// SIMATIC STEP 7 (V5.x) project My_project_Adrian
// CPU: CPU 315-2 DP
// station: P_ADR_BUS
// station: Hardware
// station: Test_station
// station: P_ADR_BUS
// station: Configuration
// program: S7 Program(1)
// program: Day1

SYMBOL_TABLE
"Counter_Bay_1"	C 1	COUNTER	// Part counter for Bay 1
"Counter_Bay_2"	C 2	COUNTER	// Part counter for Bay 2
"Counter_Bay_3"	C 3	COUNTER	// Part counter for Bay 3
"Inst_DB_Bay_1_Counter"	DB 1	SFB 0
"Inst_DB_Bay_2_Counter"	DB 2	SFB 0
"Inst_DB_Bay_3_Counter"	DB 3	SFB 0
"Inst_DB_Belt_Fault"	DB 4	SFB 4
"DB_Data_Backup"	DB 10	DB 10	// Saves the production data every minute
"Instance_FB11"	DB 11	FB 11	// Instance DB for FB11
"Instance_FB12"	DB 12	FB 12	// Instance DB for FB12
"Instance_FB16"	DB 16	FB 16	// Instance DB for FB16
"Instance_FB18"	DB 18	FB 18	// Instance DB for FB 18
"DB_Weight_Values"	DB 30	DB 30
"Instance_FB42"	DB 42	FB 42	// Instance DB for FB42
"Instance_FB44"	DB 44	FB 44	// Instance DB for FB44
"DB_Data"	DB 50	DB 50	// Stores Data for FB42: MM420 Communication
"DB_LED_Status"	DB 51	DB 51	// Stores CPU LED Status
"DB_Diagnostic_data"	DB 86	DB 86	// Stores Profibus DP Slave errors
"DB_Area_Pointer"	DB 88	DB 88	// Stores HMI Area pointers
"DB_edge_detection"	DB 100	DB 100	// Stores edge detection flags
"FB_Running_light"	FB 11	FB 11	// Running light over 1 byte
"FB_Save_weight"	FB 12	FB 12
"FB_Conveyor"	FB 16	FB 16
"FB_Statistic"	FB 18	FB 18
"FB_MM420_PKW"	FB 42	FB 42	// shows PKW mechanism
"FB_MM420"	FB 44	FB 44	// Communciation with Micromaster
"FC_DT_TOD"	FC 8	FC 8	// DT to TOD
"FC_Supply_area_pointer"	FC 12	FC 12	// supply of the HMI area pointer
"FC_Signalization"	FC 14	FC 14	// Signalization
"FC_Modes"	FC 15	FC 15	// Mode selection
"FC_Conveyor"	FC 16	FC 16	// Control logic for conveyor belt
"FC_Statistic"	FC 18	FC 18	// Count parts
"FC_Production_Display"	FC 19	FC 19	// Display production data
"FC_Diagnostic"	FC 51	FC 51	// evaluation of SZL-sublists
"FC_Scale_Analog_value"	FC 105	FC 105	// Scaling block for analog value
"Heater_Timer"	FC 119	FC 119	// Activation of heater depending upon time of day
"T00 Start"	I 0.0	BOOL	// Pushbutton - System ON
"T01 Stop"	I 0.1	BOOL	// Pushbutton - System OFF
"T02 Jog right"	I 0.2	BOOL	// Pushbutton - Jog conveyor motor right
"T03 Jog left"	I 0.3	BOOL	// Pushbutton - Jog conveyor motor left
"T04 Auto/Man"	I 0.4	BOOL	// Mode selector switch Man/Auto 0""/""1""""
"T05 Accept_Mode"	I 0.5	BOOL	// Pushbutton - Accept mode selection
"T06 Ack. Faults"	I 0.6	BOOL	// Fault Acknowledgement
"T07 Delete Memory"	I 0.7	BOOL	// Deletes the Statistic Memory
"T10 Ack_Fault"	I 1.0	BOOL	// Fault acknowledgement switch
"Analog_Store_Start"	I 1.5	BOOL	// Initiate storage of analog values into DB30
"T16_Ack_Analog_Alarm"	I 1.6	BOOL	// Reset analog HI/LO alarm
"T17_Acknowledge_Startup"	I 1.7	BOOL	// Pushbutton for startup acknowledgement
"LB1"	I 8.0	BOOL	// Light barrier at conveyor end
"T_PB1"	I 8.1	BOOL	// Acknowledge PB at Bay 1
"T_PB2"	I 8.2	BOOL	// Acknowledge PB at Bay 2
"T_PB3"	I 8.3	BOOL	// Acknowledge PB at Bay 3
"T_PB4"	I 8.4	BOOL	// Acknowledge PB at Bay 4
"BAY1"	I 8.5	BOOL	// Proximity Switch 01 for Bay1 (INI1)
"BAY2"	I 8.6	BOOL	// Proximity Switch 02 for Bay2 (INI2)
"BAY3"	I 8.7	BOOL	// Proximity Switch 03 for Bay3 (INI3)
"LB_ET"	I 88.0	BOOL
"T_PB1_ET"	I 88.1	BOOL
"T_PB2_ET"	I 88.2	BOOL
"T_PB3_ET"	I 88.3	BOOL
"T_PB4_ET"	I 88.4	BOOL
"BAY1_ET"	I 88.5	BOOL	// Proximity Switch 01 for Bay1 (INI1)
"BAY2_ET"	I 88.6	BOOL	// Proximity Switch 02 for Bay2 (INI2)
"BAY3_ET"	I 88.7	BOOL	// Proximity Switch 03 for Bay3 (INI3)
"IW_BCD"	IW 2	WORD	// BCD Thumbwheel, presets
"Always_Off"	M 0.0	BOOL	// Bit reset in OB100 at start-up
"Always_On"	M 0.1	BOOL	// Bit set in OB100 at start-up
"M_Flash_10Hz"	M 10.0	BOOL	// Memory bit - flashing frequency 10Hz
"M_Flash_2Hz"	M 10.3	BOOL	// Memory bit - flashing frequency 2Hz
"Delay_lockout"	M 14.0	BOOL	// Lockout conveyor movement after 6 seconds
"K_LT_Manual_Mode"	M 16.0	BOOL	// Conveyor runs in Manual mode
"K_LT_Auto_Mode"	M 16.1	BOOL	// Conveyor runs in Auto mode
"M_Motor_ON"	M 31.0	BOOL	// Request: Motor On
"M_Weight_OK"	M 35.0	BOOL	// Weight value is within tolerance
"M_Analog_module_error"	M 40.0	BOOL
"M_Motor_Stop"	M 46.0	BOOL	// Motor stop PB on HMI screen
"Weight_OK_Edge"	M 50.3	BOOL	// Edge storage bit for weight within tolerance message
"Weight_Not_OK_Edge"	M 50.4	BOOL	// Edge storage bit for weight outside tolerance message
"Weight_Scaled_REAL"	MD 70	REAL	// Current weight on the scale (REAL)
"Frequency_Required"	MD 130	REAL	// Enter required frequency setpoint
"Ramp_Up_Time"	MD 136	REAL	// Ramp up time value in seconds
"Ramp_Down_Time"	MD 140	REAL	// Ramp down time value in seconds
"Motor_Request"	MW 44	INT	// Command list number from HMI screen
"Quantity_Bay_1"	MW 100	INT	// Number of parts counted at Bay 1
"Quantity_Bay_2"	MW 102	INT	// Number of parts counted at Bay 2
"Quantity_Bay_3"	MW 104	INT	// Number of parts counted at Bay 3
"Total_Quantity"	MW 106	INT	// Sum of all parts counted
"Utilisation_Bay_1"	MW 110	INT	// % utilisation of bay 1
"Utilisation_Bay_2"	MW 112	INT	// % utilisation of bay 2
"Utilisation_Bay_3"	MW 114	INT	// % utilisation of bay 3
"Parameter_Number"	MW 134	INT	// Enter number of parameter to change
"CYCL_EXC"	OB 1	OB 1	// Cycle Execution
"OB_Time_Interrupt"	OB 10	OB 10
"OB_Check Weight"	OB 35	OB 35
"OB_Hardware_Interrupt"	OB 40	OB 40
"I/O_FLT1"	OB 82	OB 82	// I/O Point Fault 1
"OB_RACK_FLT"	OB 86	OB 86	// Loss of Rack Fault
"OB_Startup"	OB 100	OB 100	// automatic or manual restart
"PROG_ERR"	OB 121	OB 121	// Programming Error
"OB_Periph_Error"	OB 122	OB 122
"Status_Word_MM420"	PIW 256	WORD	// Status word from MM420 drive (feedback)
"Actual_Speed_MM420"	PIW 258	WORD	// Actual speed from MM420 drive (feedback)
"Analog_Channel_1"	PIW 304	INT	// Analog channel 1 (Potentiometer)
"Control_Word_MM420"	PQW 256	WORD	// Control word for the MM420 AC drive
"Setpoint_Speed_MM420"	PQW 258	WORD	// Setpoint speed for the MM420
"L_Belt_fault"	Q 4.0	BOOL	// Indicator light - conveyor belt fault condition
"L_SYSTEM"	Q 4.1	BOOL	// Indicator light - System ON
"L_Mode_MANUAL"	Q 4.2	BOOL	// Indicator light - MANUAL Mode ON
"L_Mode_AUTO"	Q 4.3	BOOL	// Indicator light - AUTO Mode ON
"L_Restart_M"	Q 4.5	BOOL	// Indicator light, manual restart
"L_Restart_A"	Q 4.6	BOOL	// Indicator light, auto restart
"L_Weight_not_okay"	Q 5.1	BOOL	// Indicator - weight not within tolerance
"L_Analog_Limit_Alarm"	Q 5.2	BOOL	// Analog channel has exceeded voltage limits
"Heater"	Q 5.3	BOOL	// Heater
"L_Bay1"	Q 8.1	BOOL	// Indicator light - Bay 1 (H1)
"L_Bay2"	Q 8.2	BOOL	// Indicator light - Bay 2 (H2)
"L_Bay3"	Q 8.3	BOOL	// Indicator light - Bay 3 (H3)
"L4_Preassembly"	Q 8.4	BOOL	// Indicator light - Preassembly (H4)
"K_RT"	Q 8.5	BOOL	// Contactor for Conveyor Belt move RIGHT
"K_LT"	Q 8.6	BOOL	// Contactor for Conveyor Belt move LEFT
"Horn"	Q 8.7	BOOL	// Signal on Conveyor
"L_Bay1_ET"	Q 88.1	BOOL	// Indicator light - Bay 1 (H1) into ET200S
"L_Bay2_ET"	Q 88.2	BOOL	// Indicator light - Bay 2 (H2) into ET200S
"L_Bay3_ET"	Q 88.3	BOOL	// Indicator light - Bay 3 (H3) into ET200S
"L4_Preassembly_ET"	Q 88.4	BOOL	// Indicator light - Preassembly (H4) into ET200S
"K_RT_ET"	Q 88.5	BOOL	// Contactor for Conveyor Belt move RIGHT into ET200S
"K_LT_ET"	Q 88.6	BOOL	// Contactor for Conveyor Belt move LEFT into ET200S
"Horn_ET"	Q 88.7	BOOL	// Signal on Conveyor into ET200S
"Running_Lights"	QB 8	BYTE	// Output LED's running indicate start-up has occured
"MM420_PZD"	QD 56	DWORD	// Control and main setpoint of MM420
"QW_Display"	QW 6	WORD	// Binary Coded Decimal (BCD) number display
"CTU"	SFB 0	SFB 0	// Count Up
"TON"	SFB 4	SFB 4	// Generate an On Delay
"TOF"	SFB 5	SFB 5	// Generate an Off Delay
"READ_CLK"	SFC 1	SFC 1	// Read System Clock
"DPRD_DAT"	SFC 14	SFC 14	// Read Consistent Data of a Standard DP Slave
"DPWR_DAT"	SFC 15	SFC 15	// Write Consistent Data to a Standard DP Slave
"BLKMOV"	SFC 20	SFC 20	// Copy Variables
"FILL"	SFC 21	SFC 21	// Initialize a Memory Area
"STP"	SFC 46	SFC 46	// Change the CPU to STOP
"RDSYSST"	SFC 51	SFC 51	// Read a System Status List or Partial List
"WR_USMSG"	SFC 52	SFC 52	// Write a User-Defined Diagnostic Event to the Diagnostic Buffer
"Right_Lockout_Timer"	T 1	TIMER	// 2 s lockout timer for right direction
"Left_Lockout_Timer"	T 2	TIMER	// 2 s lockout timer for left direction
"SD_Runtime_error"	T 14	TIMER	// Transport monitoring
"SD_Startup_delay"	T 16	TIMER	// Conveyor starts in Auto mode after a delay
"CPU_LED_Record"	UDT 51	UDT 51	// CPU LED information
"Conveyor_Model"	VAT 1	
"VAT_18"	VAT 2	
"VAT_FB42"	VAT 3	
END_SYMBOL_TABLE

FUNCTION_BLOCK "FB_Running_light"	// FB 11
VERSION : 0.1
VAR_INPUT
  Flash_frequency : BOOL ;
  Restart : BOOL ;
END_VAR
VAR_OUTPUT
  Running_light : BYTE ;
END_VAR
VAR
  EM_flash : BOOL ;
  EM_restart : BOOL ;
END_VAR
BEGIN
NETWORK
TITLE =
      A     #Restart;
      FP    #EM_restart;
      JCN   next;
      L     1;
      T     #Running_light;
NETWORK
TITLE =
next: A     #Restart;
      JCN   end;
      A     #Flash_frequency;
      FP    #EM_flash;
      JCN   end;
      L     #Running_light;
      SLW   1;
      L     128;
      >I;
      TAK;
      JCN   rett;
      L     1;
rett: T     #Running_light;
end:  NOP   0;
END_FUNCTION_BLOCK

FUNCTION "FC_Signalization" : VOID	// FC 14
VERSION : 0.1
BEGIN
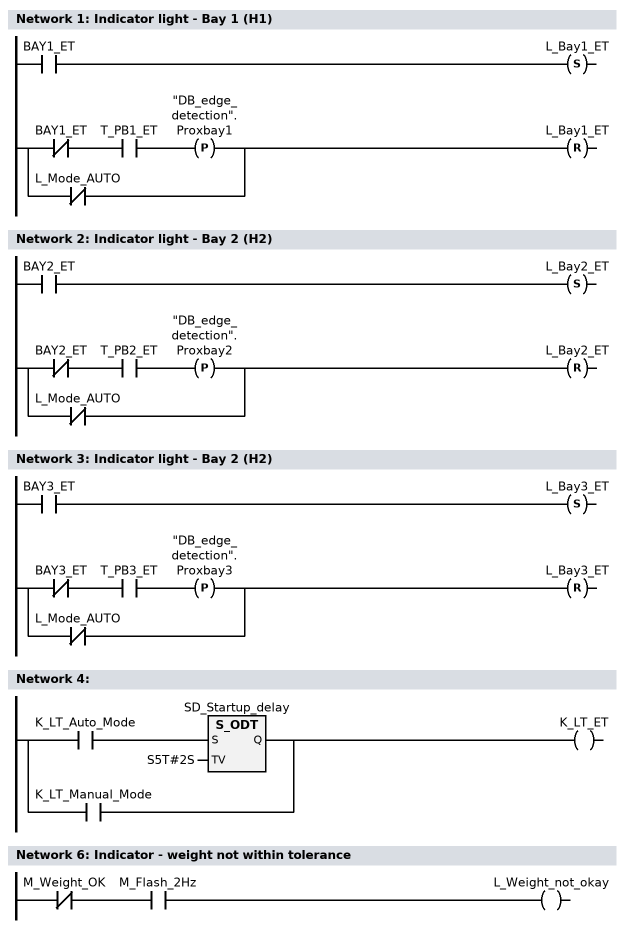
NETWORK
TITLE = Indicator light - Bay 1 (H1)
      A     "BAY1_ET";
      S     "L_Bay1_ET";
      A(;
      AN    "BAY1_ET";
      A(;
      A     "T_PB1_ET";
      BLD   100;
      FP    "DB_edge_detection".Proxbay1;
      );
      ON    "L_Mode_AUTO";
      );
      R     "L_Bay1_ET";
      NOP   0;
NETWORK
TITLE = Indicator light - Bay 2 (H2)
      A     "BAY2_ET";
      S     "L_Bay2_ET";
      A(;
      AN    "BAY2_ET";
      A(;
      A     "T_PB2_ET";
      BLD   100;
      FP    "DB_edge_detection".Proxbay2;
      );
      ON    "L_Mode_AUTO";
      );
      R     "L_Bay2_ET";
      NOP   0;
NETWORK
TITLE = Indicator light - Bay 2 (H2)
      A     "BAY3_ET";
      S     "L_Bay3_ET";
      A(;
      AN    "BAY3_ET";
      A(;
      A     "T_PB3_ET";
      BLD   100;
      FP    "DB_edge_detection".Proxbay3;
      );
      ON    "L_Mode_AUTO";
      );
      R     "L_Bay3_ET";
      NOP   0;
NETWORK
TITLE =
      O(;
      A     "K_LT_Auto_Mode";
      L     S5T#2S;
      SD    "SD_Startup_delay";
      NOP   0;
      NOP   0;
      NOP   0;
      A     "SD_Startup_delay";
      );
      O     "K_LT_Manual_Mode";
      =     "K_LT_ET";
NETWORK
TITLE =
      A(;
      A(;
      A     "K_LT_ET";
      A     "L_Restart_A";
      L     S5T#6S;
      SD    "SD_Runtime_error";
      NOP   0;
      NOP   0;
      NOP   0;
      A     "SD_Runtime_error";
      );
      S     "Delay_lockout";
      A(;
      A     "T10 Ack_Fault";
      BLD   100;
      FP    "DB_edge_detection".UNNAMED;
      );
      R     "Delay_lockout";
      A     "Delay_lockout";
      );
      A     "M_Flash_2Hz";
      =     "L_Belt_fault";
NETWORK
TITLE = Indicator - weight not within tolerance
      AN    "M_Weight_OK";
      A     "M_Flash_2Hz";
      =     "L_Weight_not_okay";
END_FUNCTION

FUNCTION "FC_Modes" : VOID	// FC 15
VERSION : 0.1
BEGIN
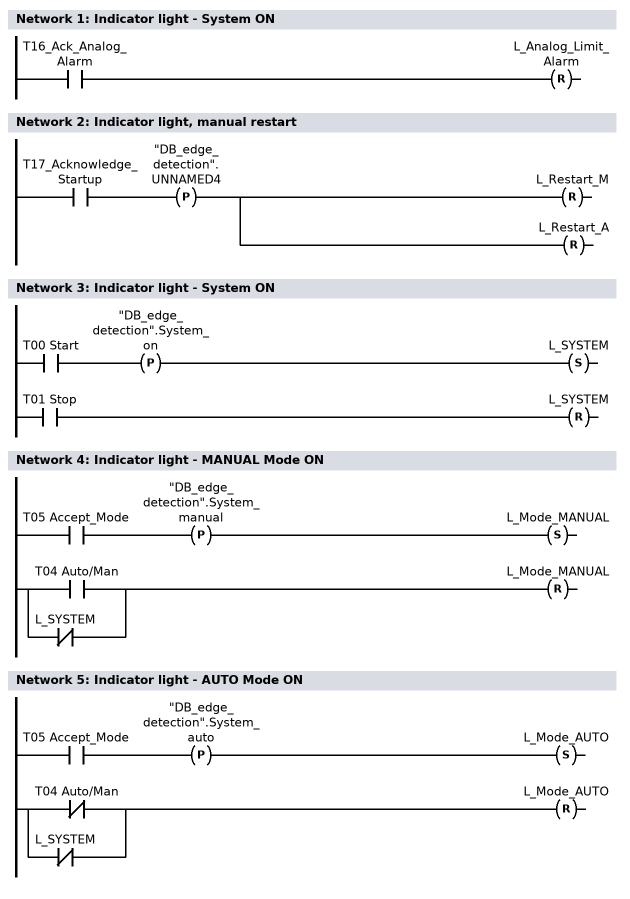
NETWORK
TITLE = Indicator light - System ON
      A     "T16_Ack_Analog_Alarm";
      R     "L_Analog_Limit_Alarm";
NETWORK
TITLE = Indicator light, manual restart
      A     "T17_Acknowledge_Startup";
      BLD   100;
      FP    "DB_edge_detection".UNNAMED4;
      R     "L_Restart_M";
      R     "L_Restart_A";
NETWORK
TITLE = Indicator light - System ON
      A     "T00 Start";
      FP    "DB_edge_detection".System_on;
      S     "L_SYSTEM";
      A     "T01 Stop";
      R     "L_SYSTEM";
      NOP   0;
NETWORK
TITLE = Indicator light - MANUAL Mode ON
      A     "T05 Accept_Mode";
      FP    "DB_edge_detection".System_manual;
      S     "L_Mode_MANUAL";
      A(;
      O     "T04 Auto/Man";
      ON    "L_SYSTEM";
      );
      R     "L_Mode_MANUAL";
      NOP   0;
NETWORK
TITLE = Indicator light - AUTO Mode ON
      A     "T05 Accept_Mode";
      FP    "DB_edge_detection".System_auto;
      S     "L_Mode_AUTO";
      A(;
      ON    "T04 Auto/Man";
      ON    "L_SYSTEM";
      );
      R     "L_Mode_AUTO";
      NOP   0;
END_FUNCTION

FUNCTION "FC_Conveyor" : VOID	// FC 16
VERSION : 0.1
BEGIN
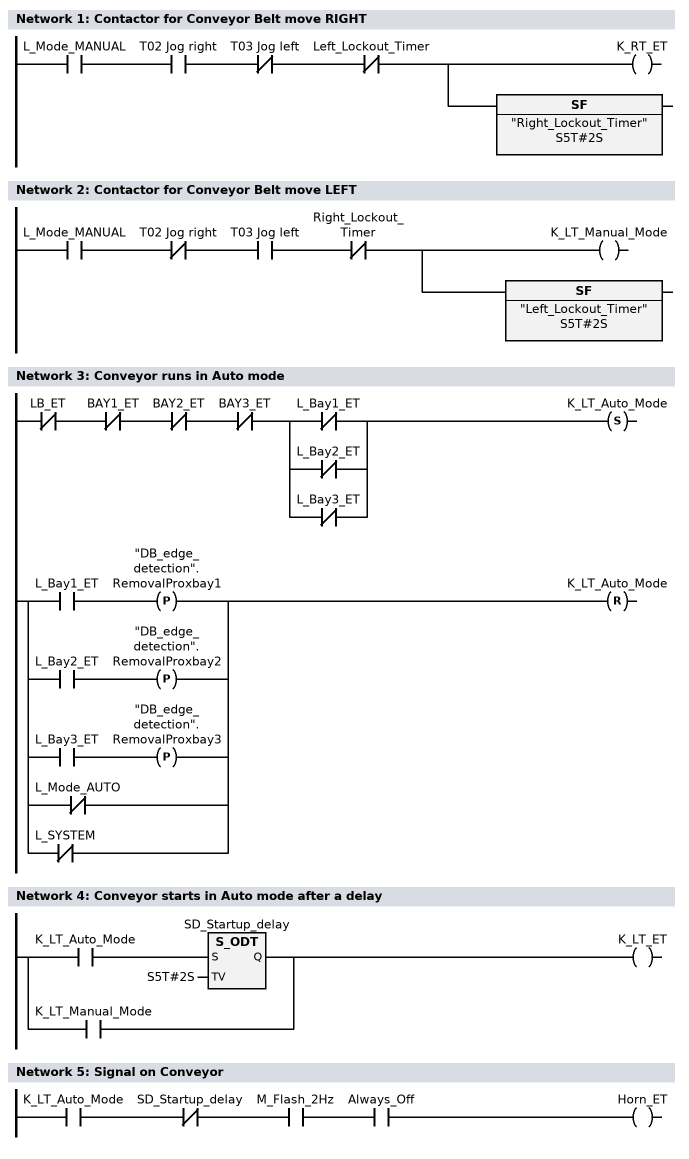
NETWORK
TITLE = Contactor for Conveyor Belt move RIGHT
      A     "L_Mode_MANUAL";
      A     "T02 Jog right";
      AN    "T03 Jog left";
      AN    "Left_Lockout_Timer";
      =     "K_RT_ET";
      L     S5T#2S;
      SF    "Right_Lockout_Timer";
NETWORK
TITLE = Contactor for Conveyor Belt move LEFT
      A     "L_Mode_MANUAL";
      AN    "T02 Jog right";
      A     "T03 Jog left";
      AN    "Right_Lockout_Timer";
      =     "K_LT_Manual_Mode";
      L     S5T#2S;
      SF    "Left_Lockout_Timer";
NETWORK
TITLE = Conveyor runs in Auto mode
      AN    "LB_ET";
      AN    "BAY1_ET";
      AN    "BAY2_ET";
      AN    "BAY3_ET";
      A(;
      ON    "L_Bay1_ET";
      ON    "L_Bay2_ET";
      ON    "L_Bay3_ET";
      );
      S     "K_LT_Auto_Mode";
      A(;
      A     "L_Bay1_ET";
      FP    "DB_edge_detection".RemovalProxbay1;
      O(;
      A     "L_Bay2_ET";
      FP    "DB_edge_detection".RemovalProxbay2;
      );
      O(;
      A     "L_Bay3_ET";
      FP    "DB_edge_detection".RemovalProxbay3;
      );
      ON    "L_Mode_AUTO";
      ON    "L_SYSTEM";
      );
      R     "K_LT_Auto_Mode";
      NOP   0;
NETWORK
TITLE = Conveyor starts in Auto mode after a delay
      O(;
      A     "K_LT_Auto_Mode";
      L     S5T#2S;
      SD    "SD_Startup_delay";
      NOP   0;
      NOP   0;
      NOP   0;
      A     "SD_Startup_delay";
      );
      O     "K_LT_Manual_Mode";
      =     "K_LT_ET";
NETWORK
TITLE = Signal on Conveyor
      A     "K_LT_Auto_Mode";
      AN    "SD_Startup_delay";
      A     "M_Flash_2Hz";
      A     "Always_Off";
      =     "Horn_ET";
END_FUNCTION

FUNCTION "FC_Statistic" : VOID	// FC 18
VERSION : 0.1
VAR_TEMP
  aux_Real : REAL ;
END_VAR
BEGIN
NETWORK
TITLE =
      A     "L_Bay1_ET";
      =     L 4.0;
      BLD   103;
      A     "T07 Delete Memory";
      FP    "DB_edge_detection".UNNAMED1;
      =     L 4.1;
      BLD   103;
      BLD   9;
      =     L 9.0;
      CDB;
      OPN   DI 1;
      TAR2  LD 5;
      A     L 4.0;
      =     DIX 0.0;
      A     L 4.1;
      =     DIX 0.1;
      LAR2  P#DBX 0.0;
      UC    "CTU";
      LAR2  LD 5;
      L     DIW 6;
      T     "Quantity_Bay_1";
      CDB;
      BLD   10;
      NOP   0;
NETWORK
TITLE = Part counter for Bay 2
      A     "L_Bay2_ET";
      =     L 4.0;
      BLD   103;
      A     "T07 Delete Memory";
      FP    "DB_edge_detection".UNNAMED2;
      =     L 4.1;
      BLD   103;
      BLD   9;
      =     L 9.0;
      CDB;
      OPN   DI 2;
      TAR2  LD 5;
      A     L 4.0;
      =     DIX 0.0;
      A     L 4.1;
      =     DIX 0.1;
      LAR2  P#DBX 0.0;
      UC    "CTU";
      LAR2  LD 5;
      L     DIW 6;
      T     "Quantity_Bay_2";
      CDB;
      BLD   10;
      NOP   0;
NETWORK
TITLE = Part counter for Bay 1
      A     "L_Bay3_ET";
      =     L 4.0;
      BLD   103;
      A     "T07 Delete Memory";
      FP    "DB_edge_detection".UNNAMED2;
      =     L 4.1;
      BLD   103;
      BLD   9;
      =     L 9.0;
      CDB;
      OPN   DI 3;
      TAR2  LD 5;
      A     L 4.0;
      =     DIX 0.0;
      A     L 4.1;
      =     DIX 0.1;
      LAR2  P#DBX 0.0;
      UC    "CTU";
      LAR2  LD 5;
      L     DIW 6;
      T     "Quantity_Bay_3";
      CDB;
      BLD   10;
      NOP   0;
NETWORK
TITLE =
      L     "Quantity_Bay_1";
      L     "Quantity_Bay_2";
      +I;
      L     "Quantity_Bay_3";
      +I;
      T     "Total_Quantity";
NETWORK
TITLE =
      L     "Total_Quantity";
      ITD;
      DTR;
      T     #aux_Real;
NETWORK
TITLE =
      L     "Total_Quantity";
      L     0;
      ==I;
      JCN   END1;
      L     0;
      T     "Utilisation_Bay_1";
      L     0;
      T     "Utilisation_Bay_1";
      T     "Utilisation_Bay_2";
      T     "Utilisation_Bay_3";
      BEU;
END1: NOP   0;
NETWORK
TITLE =
      L     "Quantity_Bay_1";
      ITD;
      DTR;
      L     1.000000e+02;
      *R;
      L     #aux_Real;
      /R;
      RND;
      T     "Utilisation_Bay_1";
NETWORK
TITLE =
      L     "Quantity_Bay_2";
      ITD;
      DTR;
      L     1.000000e+02;
      *R;
      L     #aux_Real;
      /R;
      RND;
      T     "Utilisation_Bay_2";
NETWORK
TITLE =
      L     "Quantity_Bay_3";
      ITD;
      DTR;
      L     1.000000e+02;
      *R;
      L     #aux_Real;
      /R;
      RND;
      T     "Utilisation_Bay_3";
END_FUNCTION

FUNCTION "FC_Production_Display" : VOID	// FC 19
VERSION : 0.1
VAR_INPUT
  Selection : WORD ;
END_VAR
VAR_OUTPUT
  Display : WORD ;
END_VAR
BEGIN
NETWORK
TITLE =
      L     #Selection;
      BTI;
      AW    W#16#F;
      DEC   1;
      JL    out;
      JU    bay1;
      JU    bay2;
      JU    bay3;
      JU    tot;
      JU    ut1;
      JU    ut2;
      JU    ut3;
      JU    wght;
out:  L     W#16#EEEE;
      JU    tran;
bay1: L     "Quantity_Bay_1";
      JU    anz;
bay2: L     "Quantity_Bay_2";
      JU    anz;
bay3: L     "Quantity_Bay_3";
      JU    anz;
tot:  L     "Total_Quantity";
      JU    anz;
ut1:  L     "Utilisation_Bay_1";
      JU    anz;
ut2:  L     "Utilisation_Bay_2";
      JU    anz;
ut3:  L     "Utilisation_Bay_3";
      JU    anz;
wght: L     "Weight_Scaled_REAL";
      TRUNC;
      DTB;
anz:  ITB;
tran: T     #Display;
END_FUNCTION

// FC 105: know-how protected block, not included

DATA_BLOCK "Inst_DB_Bay_1_Counter"	// DB 1
AUTHOR : SIMATIC
FAMILY : IEC_TC
VERSION : 0.0
"CTU"
BEGIN
END_DATA_BLOCK

DATA_BLOCK "Inst_DB_Bay_2_Counter"	// DB 2
AUTHOR : SIMATIC
FAMILY : IEC_TC
VERSION : 0.0
"CTU"
BEGIN
END_DATA_BLOCK

DATA_BLOCK "Inst_DB_Bay_3_Counter"	// DB 3
AUTHOR : SIMATIC
FAMILY : IEC_TC
VERSION : 0.0
"CTU"
BEGIN
END_DATA_BLOCK

DATA_BLOCK "DB_Data_Backup"	// DB 10
VERSION : 0.1
  STRUCT
   BAY : ARRAY  [1 .. 3 ] OF //counting partsfor every bay
   INT  := 0;
   Total_quantity : INT ;	//total summary
   Dummy : INT ;	//Dummy address
   Production_capacity : ARRAY  [1 .. 3 ] OF //Production capacity
   INT  := 0;
  END_STRUCT ;	
BEGIN
END_DATA_BLOCK

DATA_BLOCK "Instance_FB11"	// DB 11
VERSION : 0.0
"FB_Running_light"
BEGIN
END_DATA_BLOCK

DATA_BLOCK "DB_edge_detection"	// DB 100
VERSION : 0.1
  STRUCT
   System_on : BOOL ;
   System_manual : BOOL ;
   System_auto : BOOL ;
   Proxbay1 : BOOL ;
   Proxbay2 : BOOL ;
   Proxbay3 : BOOL ;
   RemovalProxbay1 : BOOL ;
   RemovalProxbay2 : BOOL ;
   RemovalProxbay3 : BOOL ;
   UNNAMED : BOOL ;	//Temporary placeholder variable
   UNNAMED1 : BOOL ;	//Temporary placeholder variable
   UNNAMED2 : BOOL ;	//Temporary placeholder variable
   UNNAMED3 : BOOL ;	//Temporary placeholder variable
   UNNAMED4 : BOOL ;	//Temporary placeholder variable
   UNNAMED5 : BOOL ;	//Temporary placeholder variable
   UNNAMED6 : BOOL ;	//Temporary placeholder variable
   UNNAMED7 : BOOL ;	//Temporary placeholder variable
   UNNAMED8 : BOOL ;	//Temporary placeholder variable
   UNNAMED9 : BOOL ;	//Temporary placeholder variable
   UNNAMED10 : BOOL ;	//Temporary placeholder variable
   UNNAMED11 : BOOL ;	//Temporary placeholder variable
   UNNAMED12 : BOOL ;	//Temporary placeholder variable
   UNNAMED13 : BOOL ;	//Temporary placeholder variable
   UNNAMED14 : BOOL ;	//Temporary placeholder variable
   UNNAMED15 : BOOL ;	//Temporary placeholder variable
   UNNAMED16 : BOOL ;	//Temporary placeholder variable
   UNNAMED17 : BOOL ;	//Temporary placeholder variable
   UNNAMED18 : BOOL ;	//Temporary placeholder variable
   UNNAMED19 : BOOL ;	//Temporary placeholder variable
   UNNAMED20 : BOOL ;	//Temporary placeholder variable
   UNNAMED21 : BOOL ;	//Temporary placeholder variable
   UNNAMED22 : BOOL ;	//Temporary placeholder variable
   UNNAMED23 : BOOL ;	//Temporary placeholder variable
   UNNAMED24 : BOOL ;	//Temporary placeholder variable
  END_STRUCT ;	
BEGIN
END_DATA_BLOCK

ORGANIZATION_BLOCK "CYCL_EXC"	// OB 1
TITLE = "Main Program Sweep (Cycle)"
VERSION : 0.1
VAR_TEMP
  OB1_EV_CLASS : BYTE ;	//Bits 0-3 = 1 (Coming event), Bits 4-7 = 1 (Event class 1)
  OB1_SCAN_1 : BYTE ;	//1 (Cold restart scan 1 of OB 1), 3 (Scan 2-n of OB 1)
  OB1_PRIORITY : BYTE ;	//Priority of OB Execution
  OB1_OB_NUMBR : BYTE ;	//1 (Organization block 1, OB1)
  OB1_RESERVED_1 : BYTE ;	//Reserved for system
  OB1_RESERVED_2 : BYTE ;	//Reserved for system
  OB1_PREV_CYCLE : INT ;	//Cycle time of previous OB1 scan (milliseconds)
  OB1_MIN_CYCLE : INT ;	//Minimum cycle time of OB1 (milliseconds)
  OB1_MAX_CYCLE : INT ;	//Maximum cycle time of OB1 (milliseconds)
  OB1_DATE_TIME : DATE_AND_TIME ;	//Date and time OB1 started
END_VAR
BEGIN
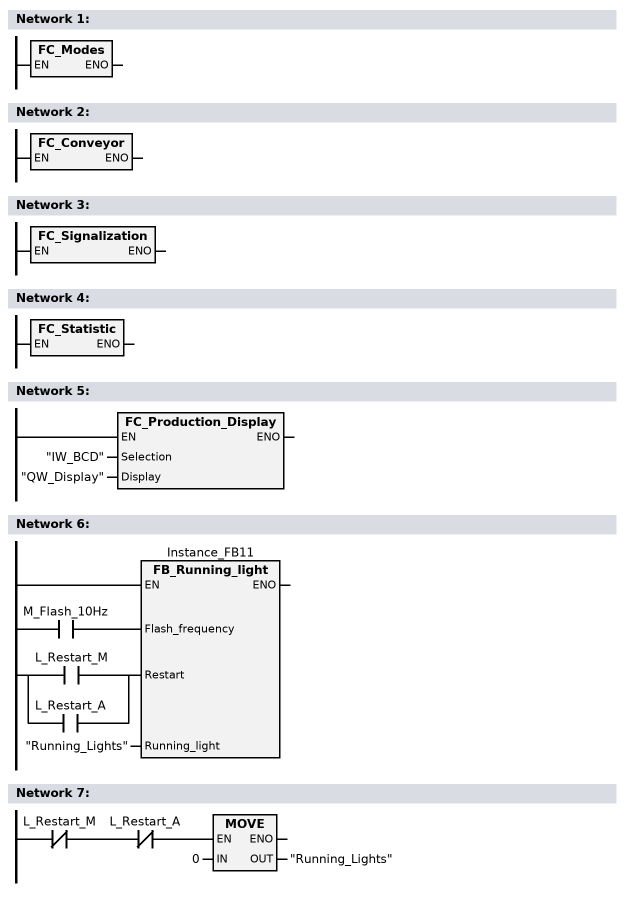
NETWORK
TITLE =
      CALL  "FC_Modes";
      NOP   0;
NETWORK
TITLE =
      CALL  "FC_Conveyor";
      NOP   0;
NETWORK
TITLE =
      CALL  "FC_Signalization";
      NOP   0;
NETWORK
TITLE =
      CALL  "FC_Statistic";
      NOP   0;
NETWORK
TITLE =
      CALL  "FC_Production_Display" (
           Selection                := "IW_BCD",
           Display                  := "QW_Display");
      NOP   0;
NETWORK
TITLE =
      A     "M_Flash_10Hz";
      =     L 20.0;
      BLD   103;
      A(;
      O     "L_Restart_M";
      O     "L_Restart_A";
      );
      =     L 20.1;
      BLD   103;
      CALL  "FB_Running_light" , "Instance_FB11" (
           Flash_frequency          := L 20.0,
           Restart                  := L 20.1,
           Running_light            := "Running_Lights");
      NOP   0;
NETWORK
TITLE =
      AN    "L_Restart_M";
      AN    "L_Restart_A";
      JNB   _001;
      L     0;
      T     "Running_Lights";
_001: NOP   0;
END_ORGANIZATION_BLOCK

ORGANIZATION_BLOCK "OB_Time_Interrupt"	// OB 10
TITLE = "Time of Day Interrupt"
VERSION : 0.1
VAR_TEMP
  OB10_EV_CLASS : BYTE ;	//Bits 0-3 = 1 (Coming event), Bits 4-7 = 1 (Event class 1)
  OB10_STRT_INFO : BYTE ;	//16#11 (OB 10 has started)
  OB10_PRIORITY : BYTE ;	//Priority of OB Execution
  OB10_OB_NUMBR : BYTE ;	//10 (Organization block 10, OB10)
  OB10_RESERVED_1 : BYTE ;	//Reserved for system
  OB10_RESERVED_2 : BYTE ;	//Reserved for system
  OB10_PERIOD_EXE : WORD ;	//Period of execution (once, per minute/hour/day/week/month/year)
  OB10_RESERVED_3 : INT ;	//Reserved for system
  OB10_RESERVED_4 : INT ;	//Reserved for system
  OB10_DATE_TIME : DATE_AND_TIME ;	//Date and time OB10 started
  Error_SFC20 : INT ;
END_VAR
BEGIN
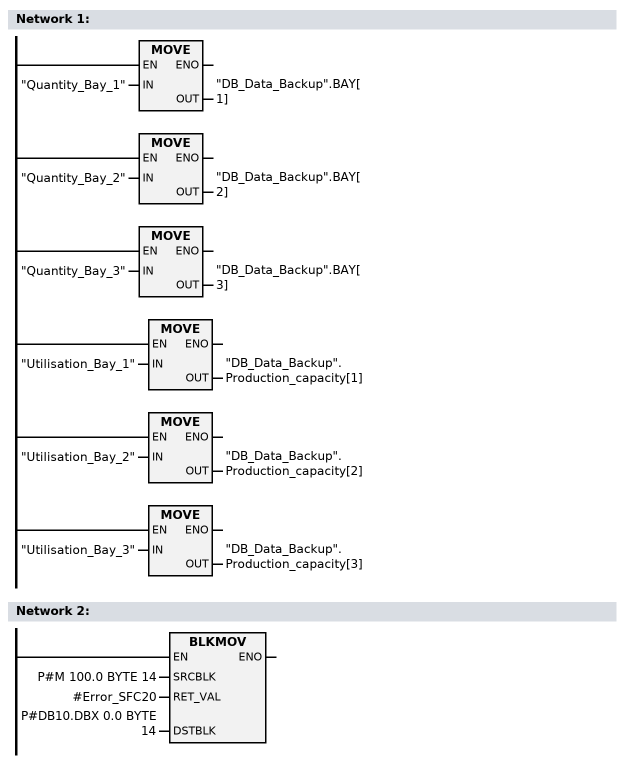
NETWORK
TITLE =
      L     "Quantity_Bay_1";
      T     "DB_Data_Backup".BAY[1];
      L     "Quantity_Bay_2";
      T     "DB_Data_Backup".BAY[2];
      L     "Quantity_Bay_3";
      T     "DB_Data_Backup".BAY[3];
      L     "Utilisation_Bay_1";
      T     "DB_Data_Backup".Production_capacity[1];
      L     "Utilisation_Bay_2";
      T     "DB_Data_Backup".Production_capacity[2];
      L     "Utilisation_Bay_3";
      T     "DB_Data_Backup".Production_capacity[3];
NETWORK
TITLE =
      CALL  "BLKMOV" (
           SRCBLK                   := P#M 100.0 BYTE 14,
           RET_VAL                  := #Error_SFC20,
           DSTBLK                   := P#DB10.DBX 0.0 BYTE 14);
      NOP   0;
END_ORGANIZATION_BLOCK

ORGANIZATION_BLOCK "OB_Check Weight"	// OB 35
TITLE = "Cyclic Interrupt"
VERSION : 0.1
VAR_TEMP
  OB35_EV_CLASS : BYTE ;	//Bits 0-3 = 1 (Coming event), Bits 4-7 = 1 (Event class 1)
  OB35_STRT_INF : BYTE ;	//16#36 (OB 35 has started)
  OB35_PRIORITY : BYTE ;	//Priority of OB Execution
  OB35_OB_NUMBR : BYTE ;	//35 (Organization block 35, OB35)
  OB35_RESERVED_1 : BYTE ;	//Reserved for system
  OB35_RESERVED_2 : BYTE ;	//Reserved for system
  OB35_PHASE_OFFSET : WORD ;	//Phase offset (msec)
  OB35_RESERVED_3 : INT ;	//Reserved for system
  OB35_EXC_FREQ : INT ;	//Frequency of execution (msec)
  OB35_DATE_TIME : DATE_AND_TIME ;	//Date and time OB35 started
  Error_FC105 : WORD ;
END_VAR
BEGIN
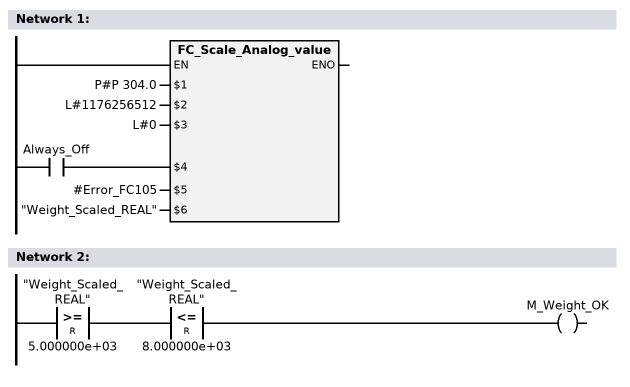
NETWORK
TITLE =
      A     "Always_Off";
      =     L 22.0;
      BLD   103;
      CALL  "FC_Scale_Analog_value" (
           $1                       := P#P 304.0,
           $2                       := L#1176256512,
           $3                       := L#0,
           $4                       := L 22.0,
           $5                       := #Error_FC105,
           $6                       := "Weight_Scaled_REAL");
      NOP   0;
NETWORK
TITLE =
      A(;
      L     "Weight_Scaled_REAL";
      L     5.000000e+03;
      >=R;
      );
      A(;
      L     "Weight_Scaled_REAL";
      L     8.000000e+03;
      <=R;
      );
      =     "M_Weight_OK";
END_ORGANIZATION_BLOCK

ORGANIZATION_BLOCK "OB_Hardware_Interrupt"	// OB 40
TITLE = "Hardware Interrupt"
VERSION : 0.1
VAR_TEMP
  OB40_EV_CLASS : BYTE ;	//Bits 0-3 = 1 (Coming event), Bits 4-7 = 1 (Event class 1)
  OB40_STRT_INF : BYTE ;	//16#41 (OB 40 has started)
  OB40_PRIORITY : BYTE ;	//Priority of OB Execution
  OB40_OB_NUMBR : BYTE ;	//40 (Organization block 40, OB40)
  OB40_RESERVED_1 : BYTE ;	//Reserved for system
  OB40_IO_FLAG : BYTE ;	//16#54 (input module), 16#55 (output module)
  OB40_MDL_ADDR : WORD ;	//Base address of module initiating interrupt
  OB40_POINT_ADDR : DWORD ;	//Interrupt status of the module
  OB40_DATE_TIME : DATE_AND_TIME ;	//Date and time OB40 started
END_VAR
BEGIN
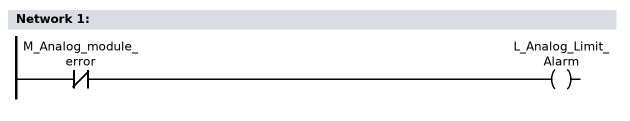
NETWORK
TITLE =
      AN    "M_Analog_module_error";
      =     "L_Analog_Limit_Alarm";
END_ORGANIZATION_BLOCK

ORGANIZATION_BLOCK "OB_Startup"	// OB 100
TITLE = "Complete Restart"
VERSION : 0.1
VAR_TEMP
  OB100_EV_CLASS : BYTE ;	//16#13, Event class 1, Entering event state, Event logged in diagnostic buffer
  OB100_STRTUP : BYTE ;	//16#81/82/83/84 Method of startup
  OB100_PRIORITY : BYTE ;	//Priority of OB Execution
  OB100_OB_NUMBR : BYTE ;	//100 (Organization block 100, OB100)
  OB100_RESERVED_1 : BYTE ;	//Reserved for system
  OB100_RESERVED_2 : BYTE ;	//Reserved for system
  OB100_STOP : WORD ;	//Event that caused CPU to stop (16#4xxx)
  OB100_STRT_INFO : DWORD ;	//Information on how system started
  OB100_DATE_TIME : DATE_AND_TIME ;	//Date and time OB100 started
END_VAR
BEGIN
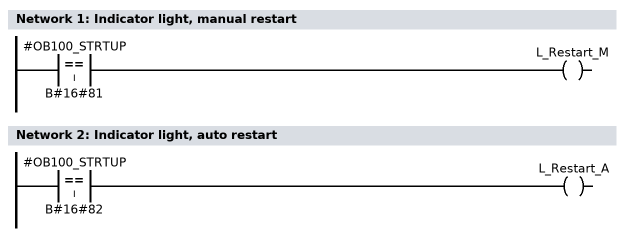
NETWORK
TITLE = Indicator light, manual restart
      L     #OB100_STRTUP;
      L     B#16#81;
      ==I;
      =     "L_Restart_M";
NETWORK
TITLE = Indicator light, auto restart
      L     #OB100_STRTUP;
      L     B#16#82;
      ==I;
      =     "L_Restart_A";
END_ORGANIZATION_BLOCK

ORGANIZATION_BLOCK "PROG_ERR"	// OB 121
TITLE = "Programming Error"
VERSION : 0.1
VAR_TEMP
  OB121_EV_CLASS : BYTE ;	//16#25, Event class 2, Entering event state, Internal fault event
  OB121_SW_FLT : BYTE ;	//16#XX Software programming fault
  OB121_PRIORITY : BYTE ;	//Priority of OB Execution
  OB121_OB_NUMBR : BYTE ;	//121 (Organization block 121, OB121)
  OB121_BLK_TYPE : BYTE ;	//16#88/8A/8B/8C/8E Type of block fault occured in
  OB121_RESERVED_1 : BYTE ;	//Reserved for system
  OB121_FLT_REG : WORD ;	//16#XX Specific register that caused fault
  OB121_BLK_NUM : WORD ;	//Number of block that programming fault occured in
  OB121_PRG_ADDR : WORD ;	//Address in block where programming fault occured
  OB121_DATE_TIME : DATE_AND_TIME ;	//Date and time OB121 started
END_VAR
BEGIN
// (block stored without names or comments; labels and parameter names are numbered)
END_ORGANIZATION_BLOCK

SYMBOL_TABLE
"Counter_Bay_1"	C 1	COUNTER	// Part counter for Bay 1
"Counter_Bay_2"	C 2	COUNTER	// Part counter for Bay 2
"Counter_Bay_3"	C 3	COUNTER	// Part counter for Bay 3
"Inst_DB_Bay_1_Counter"	DB 1	SFB 0
"Inst_DB_Bay_2_Counter"	DB 2	SFB 0
"Inst_DB_Bay_3_Counter"	DB 3	SFB 0
"Inst_DB_Belt_Fault"	DB 4	SFB 4
"DB_Data_Backup"	DB 10	DB 10	// Saves the production data every minute
"Instance_FB11"	DB 11	FB 11	// Instance DB for FB11
"Instance_FB12"	DB 12	FB 12	// Instance DB for FB12
"Instance_FB16"	DB 16	FB 16	// Instance DB for FB16
"Instance_FB18"	DB 18	FB 18	// Instance DB for FB 18
"DB_Weight_Values"	DB 30	DB 30
"Instance_FB42"	DB 42	FB 42	// Instance DB for FB42
"Instance_FB44"	DB 44	FB 44	// Instance DB for FB44
"DB_Data"	DB 50	DB 50	// Stores Data for FB42: MM420 Communication
"DB_LED_Status"	DB 51	DB 51	// Stores CPU LED Status
"DB_Diagnostic_data"	DB 86	DB 86	// Stores Profibus DP Slave errors
"DB_Area_Pointer"	DB 88	DB 88	// Stores HMI Area pointers
"DB_edge_detection"	DB 100	DB 100	// Stores edge detection flags
"FB_Running_light"	FB 11	FB 11	// Running light over 1 byte
"FB_Save_weight"	FB 12	FB 12
"FB_Conveyor"	FB 16	FB 16
"FB_Statistic"	FB 18	FB 18
"FB_MM420_PKW"	FB 42	FB 42	// shows PKW mechanism
"FB_MM420"	FB 44	FB 44	// Communciation with Micromaster
"FC_DT_TOD"	FC 8	FC 8	// DT to TOD
"FC_Supply_area_pointer"	FC 12	FC 12	// supply of the HMI area pointer
"FC_Signalization"	FC 14	FC 14	// Signalization
"FC_Modes"	FC 15	FC 15	// Mode selection
"FC_Conveyor"	FC 16	FC 16	// Control logic for conveyor belt
"FC_Statistic"	FC 18	FC 18	// Count parts
"FC_Production_Display"	FC 19	FC 19	// Display production data
"FC_Diagnostic"	FC 51	FC 51	// evaluation of SZL-sublists
"FC_Scale_Analog_value"	FC 105	FC 105	// Scaling block for analog value
"Heater_Timer"	FC 119	FC 119	// Activation of heater depending upon time of day
"T00 Start"	I 0.0	BOOL	// Pushbutton - System ON
"T01 Stop"	I 0.1	BOOL	// Pushbutton - System OFF
"T02 Jog right"	I 0.2	BOOL	// Pushbutton - Jog conveyor motor right
"T03 Jog left"	I 0.3	BOOL	// Pushbutton - Jog conveyor motor left
"T04 Auto/Man"	I 0.4	BOOL	// Mode selector switch Man/Auto 0""/""1""""
"T05 Accept_Mode"	I 0.5	BOOL	// Pushbutton - Accept mode selection
"T06 Ack. Faults"	I 0.6	BOOL	// Fault Acknowledgement
"T07 Delete Memory"	I 0.7	BOOL	// Deletes the Statistic Memory
"T10 Ack_Fault"	I 1.0	BOOL	// Fault acknowledgement switch
"Analog_Store_Start"	I 1.5	BOOL	// Initiate storage of analog values into DB30
"T16_Ack_Analog_Alarm"	I 1.6	BOOL	// Reset analog HI/LO alarm
"T17_Acknowledge_Startup"	I 1.7	BOOL	// Pushbutton for startup acknowledgement
"LB1"	I 8.0	BOOL	// Light barrier at conveyor end
"T_PB1"	I 8.1	BOOL	// Acknowledge PB at Bay 1
"T_PB2"	I 8.2	BOOL	// Acknowledge PB at Bay 2
"T_PB3"	I 8.3	BOOL	// Acknowledge PB at Bay 3
"T_PB4"	I 8.4	BOOL	// Acknowledge PB at Bay 4
"BAY1"	I 8.5	BOOL	// Proximity Switch 01 for Bay1 (INI1)
"BAY2"	I 8.6	BOOL	// Proximity Switch 02 for Bay2 (INI2)
"BAY3"	I 8.7	BOOL	// Proximity Switch 03 for Bay3 (INI3)
"LB_ET"	I 88.0	BOOL
"T_PB1_ET"	I 88.1	BOOL
"T_PB2_ET"	I 88.2	BOOL
"T_PB3_ET"	I 88.3	BOOL
"T_PB4_ET"	I 88.4	BOOL
"BAY1_ET"	I 88.5	BOOL	// Proximity Switch 01 for Bay1 (INI1)
"BAY2_ET"	I 88.6	BOOL	// Proximity Switch 02 for Bay2 (INI2)
"BAY3_ET"	I 88.7	BOOL	// Proximity Switch 03 for Bay3 (INI3)
"IW_BCD"	IW 2	WORD	// BCD Thumbwheel, presets
"Always_Off"	M 0.0	BOOL	// Bit reset in OB100 at start-up
"Always_On"	M 0.1	BOOL	// Bit set in OB100 at start-up
"M_Flash_10Hz"	M 10.0	BOOL	// Memory bit - flashing frequency 10Hz
"M_Flash_2Hz"	M 10.3	BOOL	// Memory bit - flashing frequency 2Hz
"Delay_lockout"	M 14.0	BOOL	// Lockout conveyor movement after 6 seconds
"K_LT_Manual_Mode"	M 16.0	BOOL	// Conveyor runs in Manual mode
"K_LT_Auto_Mode"	M 16.1	BOOL	// Conveyor runs in Auto mode
"M_Motor_ON"	M 31.0	BOOL	// Request: Motor On
"M_Weight_OK"	M 35.0	BOOL	// Weight value is within tolerance
"M_Analog_module_error"	M 40.0	BOOL
"M_Motor_Stop"	M 46.0	BOOL	// Motor stop PB on HMI screen
"Weight_OK_Edge"	M 50.3	BOOL	// Edge storage bit for weight within tolerance message
"Weight_Not_OK_Edge"	M 50.4	BOOL	// Edge storage bit for weight outside tolerance message
"Weight_Scaled_REAL"	MD 70	REAL	// Current weight on the scale (REAL)
"Frequency_Required"	MD 130	REAL	// Enter required frequency setpoint
"Ramp_Up_Time"	MD 136	REAL	// Ramp up time value in seconds
"Ramp_Down_Time"	MD 140	REAL	// Ramp down time value in seconds
"Motor_Request"	MW 44	INT	// Command list number from HMI screen
"Quantity_Bay 1"	MW 100	INT	// Number of parts counted at Bay 1
"Quantity_Bay_2"	MW 102	INT	// Number of parts counted at Bay 2
"Quantity_Bay_3"	MW 104	INT	// Number of parts counted at Bay 3
"Total_Quantity"	MW 106	INT	// Sum of all parts counted
"Utilisation_Bay_1"	MW 110	INT	// % utilisation of bay 1
"Utilisation_Bay_2"	MW 112	INT	// % utilisation of bay 2
"Utilisation_Bay_3"	MW 114	INT	// % utilisation of bay 3
"Parameter_Number"	MW 134	INT	// Enter number of parameter to change
"CYCL_EXC"	OB 1	OB 1	// Cycle Execution
"OB_Time_Interrupt"	OB 10	OB 10
"OB_Check Weight"	OB 35	OB 35
"OB_Hardware_Interrupt"	OB 40	OB 40
"I/O_FLT1"	OB 82	OB 82	// I/O Point Fault 1
"OB_RACK_FLT"	OB 86	OB 86	// Loss of Rack Fault
"OB_Startup"	OB 100	OB 100	// automatic or manual restart
"PROG_ERR"	OB 121	OB 121	// Programming Error
"OB_Periph_Error"	OB 122	OB 122
"Status_Word_MM420"	PIW 256	WORD	// Status word from MM420 drive (feedback)
"Actual_Speed_MM420"	PIW 258	WORD	// Actual speed from MM420 drive (feedback)
"Analog_Channel_1"	PIW 304	INT	// Analog channel 1 (Potentiometer)
"Control_Word_MM420"	PQW 256	WORD	// Control word for the MM420 AC drive
"Setpoint_Speed_MM420"	PQW 258	WORD	// Setpoint speed for the MM420
"L_Belt_fault"	Q 4.0	BOOL	// Indicator light - conveyor belt fault condition
"L_SYSTEM"	Q 4.1	BOOL	// Indicator light - System ON
"L_Mode_MANUAL"	Q 4.2	BOOL	// Indicator light - MANUAL Mode ON
"L_Mode_AUTO"	Q 4.3	BOOL	// Indicator light - AUTO Mode ON
"L_Restart_M"	Q 4.5	BOOL	// Indicator light, manual restart
"L_Restart_A"	Q 4.6	BOOL	// Indicator light, auto restart
"L_Weight_not_okay"	Q 5.1	BOOL	// Indicator - weight not within tolerance
"L_Analog_Limit_Alarm"	Q 5.2	BOOL	// Analog channel has exceeded voltage limits
"Heater"	Q 5.3	BOOL	// Heater
"L_Bay1"	Q 8.1	BOOL	// Indicator light - Bay 1 (H1)
"L_Bay2"	Q 8.2	BOOL	// Indicator light - Bay 2 (H2)
"L_Bay3"	Q 8.3	BOOL	// Indicator light - Bay 3 (H3)
"L4_Preassembly"	Q 8.4	BOOL	// Indicator light - Preassembly (H4)
"K_RT"	Q 8.5	BOOL	// Contactor for Conveyor Belt move RIGHT
"K_LT"	Q 8.6	BOOL	// Contactor for Conveyor Belt move LEFT
"Horn"	Q 8.7	BOOL	// Signal on Conveyor
"L_Bay1_ET"	Q 88.1	BOOL	// Indicator light - Bay 1 (H1) into ET200S
"L_Bay2_ET"	Q 88.2	BOOL	// Indicator light - Bay 2 (H2) into ET200S
"L_Bay3_ET"	Q 88.3	BOOL	// Indicator light - Bay 3 (H3) into ET200S
"L4_Preassembly_ET"	Q 88.4	BOOL	// Indicator light - Preassembly (H4) into ET200S
"K_RT_ET"	Q 88.5	BOOL	// Contactor for Conveyor Belt move RIGHT into ET200S
"K_LT_ET"	Q 88.6	BOOL	// Contactor for Conveyor Belt move LEFT into ET200S
"Horn_ET"	Q 88.7	BOOL	// Signal on Conveyor into ET200S
"Running_Lights"	QB 8	BYTE	// Output LED's running indicate start-up has occured
"MM420_PZD"	QD 56	DWORD	// Control and main setpoint of MM420
"QW_Display"	QW 6	WORD	// Binary Coded Decimal (BCD) number display
"CTU"	SFB 0	SFB 0	// Count Up
"TON"	SFB 4	SFB 4	// Generate an On Delay
"TOF"	SFB 5	SFB 5	// Generate an Off Delay
"READ_CLK"	SFC 1	SFC 1	// Read System Clock
"DPRD_DAT"	SFC 14	SFC 14	// Read Consistent Data of a Standard DP Slave
"DPWR_DAT"	SFC 15	SFC 15	// Write Consistent Data to a Standard DP Slave
"BLKMOV"	SFC 20	SFC 20	// Copy Variables
"FILL"	SFC 21	SFC 21	// Initialize a Memory Area
"STP"	SFC 46	SFC 46	// Change the CPU to STOP
"RDSYSST"	SFC 51	SFC 51	// Read a System Status List or Partial List
"WR_USMSG"	SFC 52	SFC 52	// Write a User-Defined Diagnostic Event to the Diagnostic Buffer
"Right_Lockout_Timer"	T 1	TIMER	// 2 s lockout timer for right direction
"Left_Lockout_Timer"	T 2	TIMER	// 2 s lockout timer for left direction
"SD_Runtime_error"	T 14	TIMER	// Transport monitoring
"SD_Startup_delay"	T 16	TIMER	// Conveyor starts in Auto mode after a delay
"CPU_LED_Record"	UDT 51	UDT 51	// CPU LED information
"Conveyor_Model"	VAT 1	
"VAT_FB42"	VAT 3	
END_SYMBOL_TABLE

FUNCTION "FC_Signalization" : VOID	// FC 14
VERSION : 0.1
BEGIN
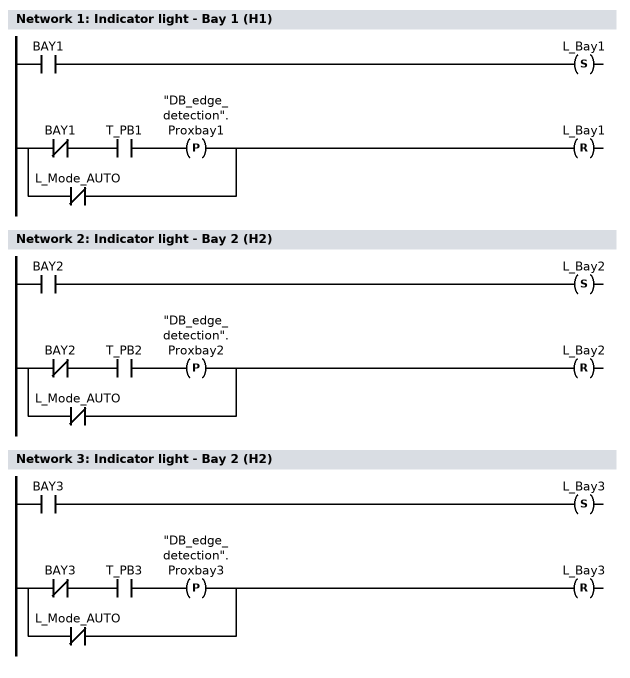
NETWORK
TITLE = Indicator light - Bay 1 (H1)
      A     "BAY1";
      S     "L_Bay1";
      A(;
      AN    "BAY1";
      A(;
      A     "T_PB1";
      BLD   100;
      FP    "DB_edge_detection".Proxbay1;
      );
      ON    "L_Mode_AUTO";
      );
      R     "L_Bay1";
      NOP   0;
NETWORK
TITLE = Indicator light - Bay 2 (H2)
      A     "BAY2";
      S     "L_Bay2";
      A(;
      AN    "BAY2";
      A(;
      A     "T_PB2";
      BLD   100;
      FP    "DB_edge_detection".Proxbay2;
      );
      ON    "L_Mode_AUTO";
      );
      R     "L_Bay2";
      NOP   0;
NETWORK
TITLE = Indicator light - Bay 2 (H2)
      A     "BAY3";
      S     "L_Bay3";
      A(;
      AN    "BAY3";
      A(;
      A     "T_PB3";
      BLD   100;
      FP    "DB_edge_detection".Proxbay3;
      );
      ON    "L_Mode_AUTO";
      );
      R     "L_Bay3";
      NOP   0;
END_FUNCTION

FUNCTION "FC_Modes" : VOID	// FC 15
VERSION : 0.1
BEGIN
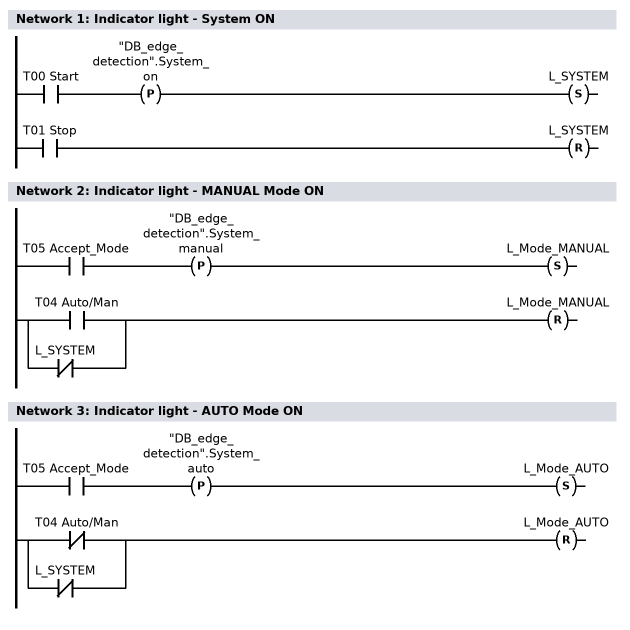
NETWORK
TITLE = Indicator light - System ON
      A     "T00 Start";
      FP    "DB_edge_detection".System_on;
      S     "L_SYSTEM";
      A     "T01 Stop";
      R     "L_SYSTEM";
      NOP   0;
NETWORK
TITLE = Indicator light - MANUAL Mode ON
      A     "T05 Accept_Mode";
      FP    "DB_edge_detection".System_manual;
      S     "L_Mode_MANUAL";
      A(;
      O     "T04 Auto/Man";
      ON    "L_SYSTEM";
      );
      R     "L_Mode_MANUAL";
      NOP   0;
NETWORK
TITLE = Indicator light - AUTO Mode ON
      A     "T05 Accept_Mode";
      FP    "DB_edge_detection".System_auto;
      S     "L_Mode_AUTO";
      A(;
      ON    "T04 Auto/Man";
      ON    "L_SYSTEM";
      );
      R     "L_Mode_AUTO";
      NOP   0;
END_FUNCTION

FUNCTION "FC_Conveyor" : VOID	// FC 16
VERSION : 0.1
BEGIN
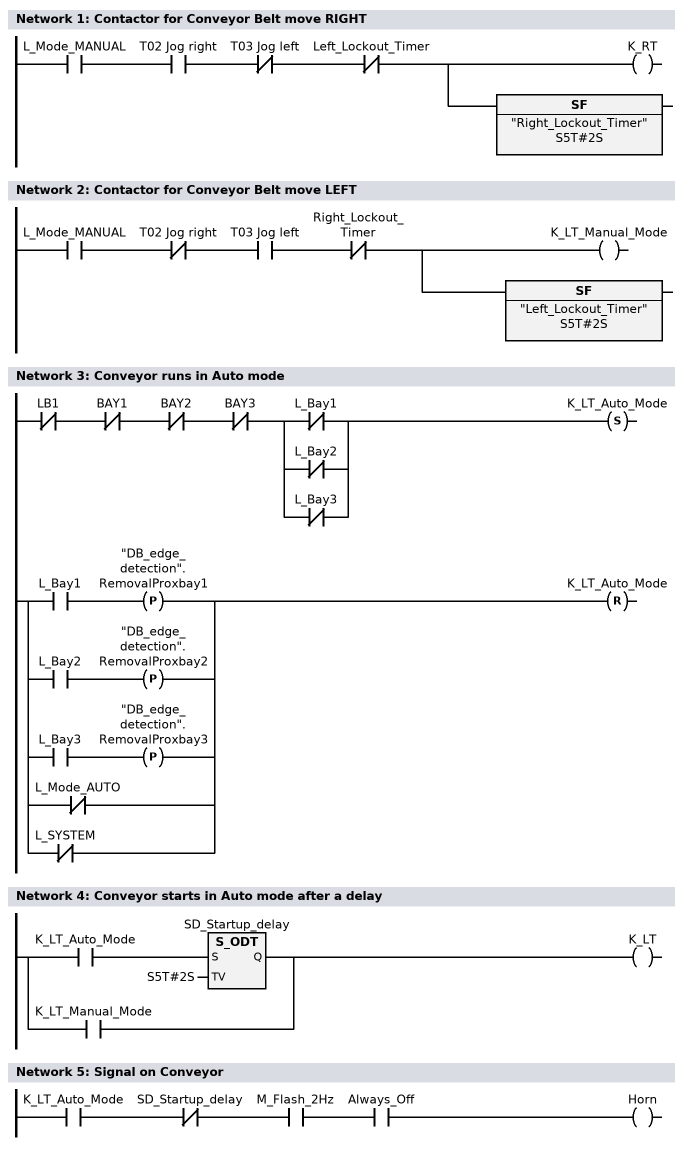
NETWORK
TITLE = Contactor for Conveyor Belt move RIGHT
      A     "L_Mode_MANUAL";
      A     "T02 Jog right";
      AN    "T03 Jog left";
      AN    "Left_Lockout_Timer";
      =     "K_RT";
      L     S5T#2S;
      SF    "Right_Lockout_Timer";
NETWORK
TITLE = Contactor for Conveyor Belt move LEFT
      A     "L_Mode_MANUAL";
      AN    "T02 Jog right";
      A     "T03 Jog left";
      AN    "Right_Lockout_Timer";
      =     "K_LT_Manual_Mode";
      L     S5T#2S;
      SF    "Left_Lockout_Timer";
NETWORK
TITLE = Conveyor runs in Auto mode
      AN    "LB1";
      AN    "BAY1";
      AN    "BAY2";
      AN    "BAY3";
      A(;
      ON    "L_Bay1";
      ON    "L_Bay2";
      ON    "L_Bay3";
      );
      S     "K_LT_Auto_Mode";
      A(;
      A     "L_Bay1";
      FP    "DB_edge_detection".RemovalProxbay1;
      O(;
      A     "L_Bay2";
      FP    "DB_edge_detection".RemovalProxbay2;
      );
      O(;
      A     "L_Bay3";
      FP    "DB_edge_detection".RemovalProxbay3;
      );
      ON    "L_Mode_AUTO";
      ON    "L_SYSTEM";
      );
      R     "K_LT_Auto_Mode";
      NOP   0;
NETWORK
TITLE = Conveyor starts in Auto mode after a delay
      O(;
      A     "K_LT_Auto_Mode";
      L     S5T#2S;
      SD    "SD_Startup_delay";
      NOP   0;
      NOP   0;
      NOP   0;
      A     "SD_Startup_delay";
      );
      O     "K_LT_Manual_Mode";
      =     "K_LT";
NETWORK
TITLE = Signal on Conveyor
      A     "K_LT_Auto_Mode";
      AN    "SD_Startup_delay";
      A     "M_Flash_2Hz";
      A     "Always_Off";
      =     "Horn";
END_FUNCTION

FUNCTION "FC_Statistic" : VOID	// FC 18
VERSION : 0.1
BEGIN
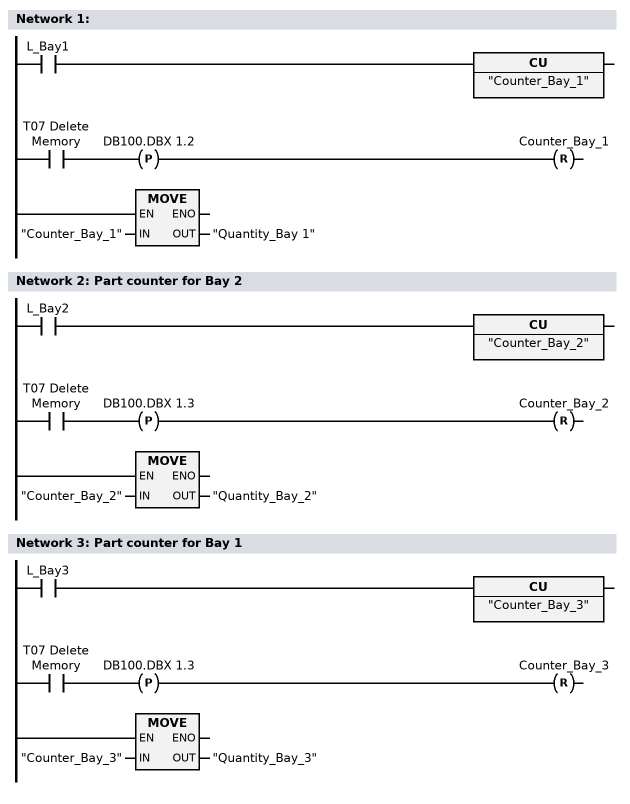
NETWORK
TITLE =
      A     "L_Bay1";
      CU    "Counter_Bay_1";
      BLD   101;
      NOP   0;
      NOP   0;
      A     "T07 Delete Memory";
      FP    DB100.DBX 1.2;
      R     "Counter_Bay_1";
      L     "Counter_Bay_1";
      T     "Quantity_Bay 1";
      NOP   0;
      NOP   0;
NETWORK
TITLE = Part counter for Bay 2
      A     "L_Bay2";
      CU    "Counter_Bay_2";
      BLD   101;
      NOP   0;
      NOP   0;
      A     "T07 Delete Memory";
      FP    DB100.DBX 1.3;
      R     "Counter_Bay_2";
      L     "Counter_Bay_2";
      T     "Quantity_Bay_2";
      NOP   0;
      NOP   0;
NETWORK
TITLE = Part counter for Bay 1
      A     "L_Bay3";
      CU    "Counter_Bay_3";
      BLD   101;
      NOP   0;
      NOP   0;
      A     "T07 Delete Memory";
      FP    DB100.DBX 1.3;
      R     "Counter_Bay_3";
      L     "Counter_Bay_3";
      T     "Quantity_Bay_3";
      NOP   0;
      NOP   0;
END_FUNCTION

DATA_BLOCK "DB_edge_detection"	// DB 100
VERSION : 0.1
  STRUCT
   System_on : BOOL ;	//Temporary placeholder variable
   System_manual : BOOL ;
   System_auto : BOOL ;
   Proxbay1 : BOOL ;
   Proxbay2 : BOOL ;
   Proxbay3 : BOOL ;
   RemovalProxbay1 : BOOL ;
   RemovalProxbay2 : BOOL ;
   RemovalProxbay3 : BOOL ;
  END_STRUCT ;	
BEGIN
END_DATA_BLOCK

ORGANIZATION_BLOCK "CYCL_EXC"	// OB 1
TITLE = "Main Program Sweep (Cycle)"
VERSION : 0.1
VAR_TEMP
  OB1_EV_CLASS : BYTE ;	//Bits 0-3 = 1 (Coming event), Bits 4-7 = 1 (Event class 1)
  OB1_SCAN_1 : BYTE ;	//1 (Cold restart scan 1 of OB 1), 3 (Scan 2-n of OB 1)
  OB1_PRIORITY : BYTE ;	//Priority of OB Execution
  OB1_OB_NUMBR : BYTE ;	//1 (Organization block 1, OB1)
  OB1_RESERVED_1 : BYTE ;	//Reserved for system
  OB1_RESERVED_2 : BYTE ;	//Reserved for system
  OB1_PREV_CYCLE : INT ;	//Cycle time of previous OB1 scan (milliseconds)
  OB1_MIN_CYCLE : INT ;	//Minimum cycle time of OB1 (milliseconds)
  OB1_MAX_CYCLE : INT ;	//Maximum cycle time of OB1 (milliseconds)
  OB1_DATE_TIME : DATE_AND_TIME ;	//Date and time OB1 started
END_VAR
BEGIN
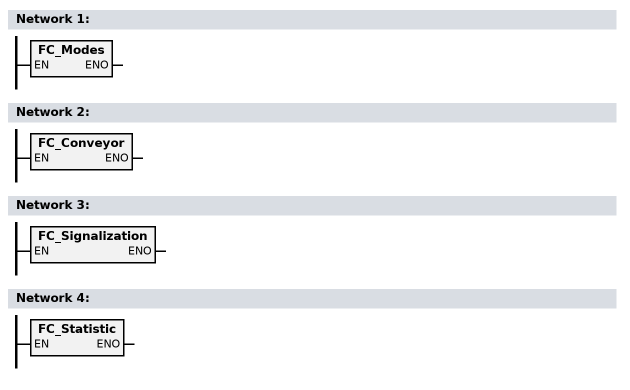
NETWORK
TITLE =
      CALL  "FC_Modes";
      NOP   0;
NETWORK
TITLE =
      CALL  "FC_Conveyor";
      NOP   0;
NETWORK
TITLE =
      CALL  "FC_Signalization";
      NOP   0;
NETWORK
TITLE =
      CALL  "FC_Statistic";
      NOP   0;
END_ORGANIZATION_BLOCK
